{attribute 'linkalways'} 
{attribute 'no_explicit_call' := 'This FB is a CLASS and must be accessed using methods or properties'}
{attribute 'enable_dynamic_creation'}
FUNCTION_BLOCK Node_F_VN_MaxElementElementwise_TcVnVector3_INT EXTENDS VisionNode
VAR
    ipContainer : _ITcVnContainer;
    aMax : _TcVnVector3_INT;
    hrPrev : _HRESULT(S_OK);
    hresult : _HRESULT(S_OK);
END_VAR

METHOD PUBLIC  Clone : I_Node
VAR
	pNode : POINTER TO Node_F_VN_MaxElementElementwise_TcVnVector3_INT;
END_VAR
pNode := __NEW(Node_F_VN_MaxElementElementwise_TcVnVector3_INT);
Clone := pNode^;
END_METHOD

METHOD FB_init : BOOL
VAR_INPUT
	bInitRetains : BOOL; // if TRUE, the retain variables are initialized (warm start / cold start)
	bInCopyCode : BOOL;  // if TRUE, the instance afterwards gets moved into the copy code (online change)
END_VAR
AddInput('ipContainer', ipContainer);
AddInput('hrPrev', hrPrev);
AddOutput('ipContainer', ipContainer);
AddOutput('aMax', aMax);
AddOutput('hresult',hresult);
END_METHOD

METHOD PROTECTED OnExecute
hresult.Value := F_VN_MaxElementElementwise_TcVnVector3_INT(
    ipContainer := ipContainer.Value,
    aMax := aMax.Value,
    hrPrev:= hrPrev.Value);
END_METHOD

METHOD PUBLIC PreExecutionCheck
VAR_INPUT
	Check : I_PreExecutionChecks;
END_VAR
Check.IsTrue(ipContainer.IsValid, 'ipContainer must be a valid container');
Check.IsTrue(ipContainer.IsType(TC_GLOBAL_CONST_LIST.ContainerType_Vector_TcVnVector3_INT), 'ipContainer contains incorrect type');
END_METHOD

END_FUNCTION_BLOCK

(* stored: Version 1.1.0.1, ProductVersion 3.1.4026.13
   POU Node_F_VN_MaxElementElementwise_TcVnVector3_INT: Id {22ae8864-6143-4326-837c-0434ba290b07}, SpecialFunc None
   Folder Constructor: Id {c45d474a-650c-405f-b6be-9fb8e8f9d411}
   Method Clone: Id {60d74211-7bb9-40ad-9426-0e8d86e604ac}
   Method FB_init: Id {8439f9f7-75f0-4b09-9535-fa569d84770c}
   Method OnExecute: Id {b2baae41-e74d-46dd-af94-63b3d2e08272}
   Method PreExecutionCheck: Id {0bba9d21-024d-45e9-b9c0-fd706adcd2f1} *)
